PROGRAM MAIN
VAR
	FilterCycle1 : FB_FILTER;  // instantie van FB
	WaterCooling1: FB_WATERCOOLING;	
	CO2_1:FB_CO2;
	LIGHT1:FB_LIGHT;
	HEATING1:FB_HEATING;	
	
END_VAR

GVL.id_TEMP_SETPOINT:=28;

IF GVL.ix_TEMPRESET THEN
	GVL.id_TEMP_SENSOR := 30;
	GVL.ix_TEMPRESET:=FALSE;
END_IF

IF GVL.ix_COOLDOWN THEN
	GVL.id_TEMP_SENSOR := GVL.id_TEMP_SENSOR -5;
	GVL.ix_COOLDOWN:=FALSE;
END_IF	

// GVL output koppelen
GVL.ox_HEATER :=HEATING1.HEATING;
GVL.ox_CO2 :=CO2_1.CO2;
GVL.ox_FILTER_WATER := FilterCycle1.FILTER_WATER;
GVL.ox_LIGHT :=LIGHT1.LIGHT;

//FUNCTIEBLOKKEN
WaterCooling1(HEATER:=GVL.ox_HEATER,TEMP_SENSOR:=GVL.id_TEMP_SENSOR);
FilterCycle1(ix_START := GVL.ix_START);
CO2_1(ix_START :=GVL.ix_START);
LIGHT1(ix_START :=GVL.ix_START);
HEATING1(ix_START:=GVL.ix_START,
TEMP:=GVL.id_TEMP_SENSOR,
SETPOINT:=GVL.id_TEMP_SETPOINT);

END_PROGRAM

(* stored: Version 1.1.0.1, ProductVersion 3.1.4024.15
   POU MAIN: Id {75683ed3-513e-4c3d-9049-ff092608163c}, SpecialFunc None *)
